{attribute 'qualified_only'}
{attribute 'strict'}
TYPE E_DataSet :
(
	SETPOINTS := 1,
	ACTUAL := 2
);
END_TYPE

(* stored: Version 1.1.0.1, ProductVersion 3.1.4024.0
   DUT E_DataSet: Id {1974b610-bddf-4616-8e97-eedade75fee5} *)
